TYPE ST_DefaultIdentityOUT1 :
STRUCT
	SKU						:STRING;
	GTIN					:STRING;
	ProductionOrder			:STRING;
	LocalProductionOrder	:STRING;
	PITCode					:STRING;
	BatchID					:STRING;
	ProductionLine			:STRING;
END_STRUCT
END_TYPE

(* stored: Version 1.1.0.1, ProductVersion 3.1.4024.13
   DUT ST_DefaultIdentityOUT1: Id {d48ea864-3649-43bf-a313-35af067236cb} *)
